Yaskawa INFORM job: R1_W68-69(-90,-90)KM-OK.JBI

/JOB
//NAME R1_W68-69(-90,-90)KM-OK
///FOLDERNAME KRIS-SCIANA
//POS
///NPOS 52,52,0,4,0,0
///TOOL 0
///POSTYPE PULSE
///PULSE
C00000=-59135,-25377,-6981,-14089,62612,-17507
C00001=-62613,-31099,-7610,-14128,60942,-21463
C00002=-59940,-5159,40679,-18119,45646,-17920
C00003=-59624,3615,52643,-19120,42998,-17213
C00004=-59501,7492,57968,-19613,41807,-16882
C00005=-59497,11001,63803,-20311,40123,-16465
C00006=-59501,10089,62300,-20126,40550,-16575
C00007=-61383,14866,67229,-19871,39625,-17199
C00008=-62013,16353,68644,-19745,39399,-17430
C00009=-61104,13358,65192,-19754,40130,-17194
C00010=-76059,4190,67286,29566,19398,-37319
C00011=-74863,5587,68510,28478,19047,-36529
C00012=-77214,-1677,58860,27807,21620,-36745
C00013=-70565,11395,57405,-1505,43209,-27686
C00014=-71720,2948,45409,-1099,46233,-28211
C00015=-49054,52400,94850,59,71875,26451
C00016=-49054,26059,47856,57,87262,26459
C00017=-49054,27038,49871,57,86525,26459
C00018=-49972,30482,54726,-129,85305,26164
C00019=-49972,31976,57659,-129,84268,26165
C00020=-49524,30460,55672,-37,84713,26308
C00021=-50449,32645,57909,-225,84457,26012
C00022=-51067,34180,59498,-350,84267,25815
C00023=-50458,32666,57930,-227,84455,26008
C00024=-50458,26424,45164,-227,89103,26000
C00025=-64210,3164,44535,-3054,77287,21763
C00026=-65385,8893,54563,-3336,74023,21486
C00027=-65855,11500,58998,-3455,72618,21383
C00028=-65850,14757,64478,-3487,70923,21432
C00029=-65778,14008,63381,-3467,71216,21447
C00030=-66632,16482,65849,-3651,70938,21198
C00031=-67176,18022,67325,-3766,70798,21038
C00032=-66605,13962,61669,-3619,72212,21167
C00033=-61181,40676,95721,-11354,75046,25122
C00034=-61844,38092,92763,-11554,75457,24900
C00035=-60614,43135,98592,-11186,74615,25320
C00036=-67045,30525,80104,-2911,78785,22235
C00037=-65957,23710,67836,-2535,82860,22462
C00038=-66976,11986,60686,-52108,68160,17724
C00039=-82575,28324,48009,-11244,75457,-6524
C00040=-76886,5805,47599,-26353,45878,17749
C00041=-66475,9175,56958,-51734,68940,17497
C00042=-66263,10146,59005,-51903,68560,17828
C00043=-96613,1823,46180,24726,37558,-4880
C00044=-85834,-7768,42641,-18506,24245,-14056
C00045=-69424,13177,60279,-31484,28536,-4386
C00046=-66302,19328,66119,-33739,29201,-2605
C00047=-66989,11978,60679,-36618,26945,7124
C00048=-66987,11980,60680,-36619,26946,7125
C00049=-66978,12004,60703,-36626,26948,7130
C00050=-66831,-18265,3169,-22895,44504,-326
C00051=-68370,-159560,-130732,-23103,44734,-299
BC00000=234960,124480,853973
BC00001=239173,128524,845479
BC00002=239173,128524,845479
BC00003=239173,128524,845479
BC00004=239173,128524,845479
BC00005=239173,128524,845479
BC00006=239173,128524,845479
BC00007=239173,128524,845479
BC00008=239173,128524,845479
BC00009=239173,128524,845479
BC00010=239173,128524,845479
BC00011=239173,128524,845479
BC00012=239173,128524,845479
BC00013=239173,128524,845479
BC00014=239173,128524,845479
BC00015=183094,164096,846547
BC00016=183094,164096,721996
BC00017=183094,164096,721996
BC00018=183094,164096,721996
BC00019=183094,164096,721996
BC00020=183094,164096,721996
BC00021=183094,164096,721996
BC00022=183094,164096,721996
BC00023=183094,164096,721996
BC00024=183094,164096,721996
BC00025=183094,164097,846551
BC00026=183094,164097,846551
BC00027=183094,164097,846551
BC00028=183094,164097,846551
BC00029=183094,164097,846551
BC00030=183094,164097,846551
BC00031=183094,164097,846551
BC00032=183094,164097,846551
BC00033=183094,164097,846551
BC00034=183094,164097,846551
BC00035=183094,164097,846551
BC00036=183094,164097,846551
BC00037=183094,164097,846551
BC00038=218908,93793,858602
BC00039=175376,88865,762723
BC00040=180813,88771,762962
BC00041=215063,101817,729636
BC00042=215063,101817,729636
BC00043=180813,88771,762962
BC00044=236761,88770,762963
BC00045=236831,88770,762964
BC00046=236831,88770,762964
BC00047=241398,88120,767024
BC00048=238054,82546,781671
BC00049=238054,82546,889206
BC00050=238054,82546,889206
BC00051=238054,117917,889206
///POSTYPE BASE
///RECTAN
///RCONF 0,0,0,0,1,0,0,0,0,0,0,0,0,0,0,0,0,0,0,0,0,0,0,0
P00006=2.006,1.622,-0.565,0.0000,0.0000,0.0000
P00021=0.073,2.058,-0.109,0.0000,0.0000,0.0000
P00022=2.006,1.622,-0.565,0.0000,0.0000,0.0000
///RCONF 0,0,0,0,0,0,0,0,0,0,0,0,0,0,0,0,0,0,0,0,0,0,0,0
P00030=-0.014,-0.768,0.131,0.0000,0.0000,0.0000
//INST
///DATE 2025/04/14 13:41
///ATTR SC,RW
///GROUP1 RB1,BS1
NOP
'r1_W68-69(-90,-90)
'Path S836 (for W508)
SFTOF
MOVJ C00000 BC00000 VJ=100.00
MOVJ C00001 BC00001 VJ=100.00
MOVJ C00002 BC00002 VJ=100.00
MOVJ C00003 BC00003 VJ=100.00
MOVL C00004 BC00004 V=60.0
REFP 3 C00005 BC00005
CALL JOB:SEARCH-R1
SET P021 P006
SFTON P021
MOVL C00006 BC00006 V=60.0
MOVL C00007 BC00007 V=60.0
REFP 3 C00008 BC00008
CALL JOB:SEARCH-R1
SET P021 P006
SFTON P021
MOVL C00009 BC00009 V=60.0
MOVL C00010 BC00010 V=60.0
REFP 3 C00011 BC00011
CALL JOB:SEARCH-R1
SET P021 P006
SFTON P021
MOVL C00012 BC00012 V=60.0
MOVL C00013 BC00013 V=100.0
MOVL C00014 BC00014 V=166.7
'Path S837 (for W508)
SFTOF
MOVL C00015 BC00015 V=1000.0
MOVL C00016 BC00016 V=1000.0
MOVL C00017 BC00017 V=100.0
MOVL C00018 BC00018 V=60.0
REFP 3 C00019 BC00019
CALL JOB:SEARCH-R1
SET P030 P006
SFTON P030
MOVL C00020 BC00020 V=60.0
MOVL C00021 BC00021 V=60.0
REFP 3 C00022 BC00022
CALL JOB:SEARCH-R1
SET P030 P006
SFTON P030
MOVL C00023 BC00023 V=60.0
MOVL C00024 BC00024 V=400.0
SFTOF
MOVL C00025 BC00025 V=166.7
MOVL C00026 BC00026 V=100.0
MOVL C00027 BC00027 V=60.0
REFP 3 C00028 BC00028
CALL JOB:SEARCH-R1
SET P022 P006
SFTON P022
MOVL C00029 BC00029 V=60.0
MOVL C00030 BC00030 V=60.0
REFP 3 C00031 BC00031
CALL JOB:SEARCH-R1
SET P022 P006
SFTON P022
MOVL C00032 BC00032 V=60.0
MOVL C00033 BC00033 V=60.0
REFP 3 C00034 BC00034
CALL JOB:SEARCH-R1
SET P022 P006
SFTON P022
MOVL C00035 BC00035 V=60.0
MOVL C00036 BC00036 V=100.0
MOVL C00037 BC00037 V=400.0
'Path W508
SFTOF
SFTON P022
CALL JOB:COFNIJ_DRUT
MOVJ C00038 BC00038 VJ=100.00
MOVJ C00039 BC00039 VJ=100.00
MOVL C00040 BC00040 V=100.0 PL=0
REFP 1 C00041 BC00041
REFP 2 C00042 BC00042
MACRO1 MJ#(0) ARGF9
ARCON
MOVL C00043 BC00043 V=10.8
SFTON P030
MOVL C00044 BC00044 V=10.8
SFTON P021
MOVL C00045 BC00045 V=10.8
MOVL C00046 BC00046 V=10.8
ARCOF
MOVL C00047 BC00047 V=100.0
MOVL C00048 BC00048 V=166.7
MOVL C00049 BC00049 V=166.7
SFTOF
MOVJ C00050 BC00050 VJ=100.00
MOVJ C00051 BC00051 VJ=100.00
END
